ABB RobotStudio station: SD_Exe01_SWorksRStudio.rsstnx

Station SD_Exe01_SWorksRStudio (saved by RobotStudio 22.3.10190.2)
Controller CRB15000_5_95_1
  mechanical unit ROB_1: CRB15000_5_95__02, 6 joints, base frame (0, 0, 0) mm
Layout (positions relative to the parent item):
  - CRB15000_5_95__02 [mechanism, from Robots\CRB15000_5_95__02.rslib] at (0, 0, 0) mm; joint values [0.1436, 0.0868, 0.8423, 1.7766, 1.4192, 2.1968] (rad or m)
  - EF_DemoTool [mechanism] at (461.55, 153.56, 331.85) mm, rotated rx -90 ry 0 rz -6.38 deg
      TCP EF_DemoTool at (0, 0, 155) mm
      links: EF_Demo
  - part_SD_01 [part] at (485.51, 347.24, 308) mm, size 71 x 71 x 39 mm
  - table_and_fixture_140 [part, from Training Objects\propeller_table.rslib] at (292.34, 222.04, 0) mm
Attachment: EF_DemoTool is attached to CRB15000_5_95__02 / Link6
Attachment: Workobject_1 is attached to part_SD_01
Attachment: Workobject_3 is attached to table_and_fixture_140
Attachment: part_SD_01 is attached to table_and_fixture_140
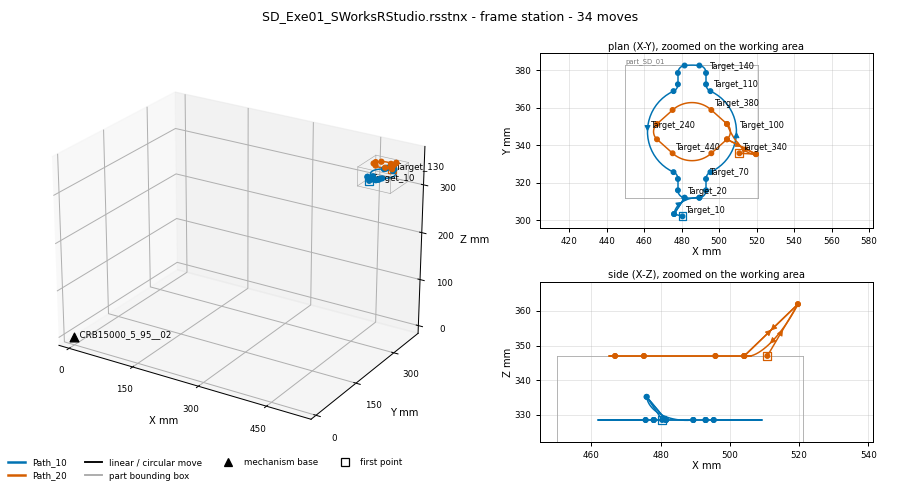
[picture p0: tool path of SD_Exe01_SWorksRStudio.rsstnx in frame station, 34 of 34 moves have a stored position in this frame; points joined in program order, loops and branches not executed]
Targets, tools, work objects and paths stored in the station, written as RAPID:
! task T_ROB1
MODULE CalibData
  PERS tooldata EF_DemoTool:=[TRUE,[[0,0,155],[1,0,0,0]],[2,[20,0,15],[1,0,0,0],0,0,0]];
  PERS wobjdata Workobject_1:=[FALSE,TRUE,"",[[485.512,347.241,308],[1,0,0,0]],[[0,0,0],[1,0,0,0]]];
  PERS wobjdata Workobject_3:=[FALSE,TRUE,"",[[485.512,347.241,308],[1,0,0,0]],[[0,0,0],[1,0,0,0]]];
ENDMODULE

! task T_ROB1
MODULE Module1
  CONST robtarget Target_10:=[[-5.055555556,-45.218263545,20.5],[0.70601133,-0.70601133,0.039344663,-0.039344663],[0,1,1,0],[9E+09,9E+09,9E+09,9E+09,9E+09,9E+09]];
  CONST robtarget Target_20:=[[-3.944444444,-35.280183645,20.5],[0.70601133,-0.70601133,0.039344663,-0.039344663],[0,1,1,0],[9E+09,9E+09,9E+09,9E+09,9E+09,9E+09]];
  CONST robtarget Target_30:=[[0,-35.5,20.5],[0.70601133,-0.70601133,0.039344663,-0.039344663],[0,1,1,0],[9E+09,9E+09,9E+09,9E+09,9E+09,9E+09]];
  CONST robtarget Target_40:=[[3.944444444,-35.280183645,20.5],[0.70601133,-0.70601133,0.039344663,-0.039344663],[0,1,1,0],[9E+09,9E+09,9E+09,9E+09,9E+09,9E+09]];
  CONST robtarget Target_50:=[[6.48142397,-33.971618352,20.5],[0.70601133,-0.70601133,0.039344663,-0.039344663],[0,1,1,0],[9E+09,9E+09,9E+09,9E+09,9E+09,9E+09]];
  CONST robtarget Target_60:=[[7.5,-31.304951685,20.5],[0.70601133,-0.70601133,0.039344663,-0.039344663],[0,1,1,0],[9E+09,9E+09,9E+09,9E+09,9E+09,9E+09]];
  CONST robtarget Target_70:=[[7.5,-25.25495001,20.5],[0.70601133,-0.70601133,0.039344663,-0.039344663],[0,1,1,0],[9E+09,9E+09,9E+09,9E+09,9E+09,9E+09]];
  CONST robtarget Target_80:=[[8.136175493,-23.090536767,20.5],[0.70601133,-0.70601133,0.039344663,-0.039344663],[0,1,1,0],[9E+09,9E+09,9E+09,9E+09,9E+09,9E+09]];
  CONST robtarget Target_90:=[[9.842342342,-21.614596855,20.5],[0.70601133,-0.70601133,0.039344663,-0.039344663],[0,1,1,0],[9E+09,9E+09,9E+09,9E+09,9E+09,9E+09]];
  CONST robtarget Target_100:=[[23.75,0,20.5],[0.70601133,-0.70601133,0.039344663,-0.039344663],[0,1,1,0],[9E+09,9E+09,9E+09,9E+09,9E+09,9E+09]];
  CONST robtarget Target_110:=[[9.842342342,21.614596855,20.5],[0.70601133,-0.70601133,0.039344663,-0.039344663],[0,1,1,0],[9E+09,9E+09,9E+09,9E+09,9E+09,9E+09]];
  CONST robtarget Target_120:=[[8.136175493,23.090536767,20.5],[0.70601133,-0.70601133,0.039344663,-0.039344663],[0,1,1,0],[9E+09,9E+09,9E+09,9E+09,9E+09,9E+09]];
  CONST robtarget Target_130:=[[7.5,25.25495001,20.5],[0.70601133,-0.70601133,0.039344663,-0.039344663],[0,1,1,0],[9E+09,9E+09,9E+09,9E+09,9E+09,9E+09]];
  CONST robtarget Target_140:=[[7.5,31.304951685,20.5],[0.70601133,-0.70601133,0.039344663,-0.039344663],[0,1,1,0],[9E+09,9E+09,9E+09,9E+09,9E+09,9E+09]];
  CONST robtarget Target_150:=[[6.48142397,33.971618352,20.5],[0.70601133,-0.70601133,0.039344663,-0.039344663],[0,1,1,0],[9E+09,9E+09,9E+09,9E+09,9E+09,9E+09]];
  CONST robtarget Target_160:=[[3.944444444,35.280183645,20.5],[0.70601133,-0.70601133,0.039344663,-0.039344663],[0,1,1,0],[9E+09,9E+09,9E+09,9E+09,9E+09,9E+09]];
  CONST robtarget Target_170:=[[0,35.5,20.5],[0.70601133,-0.70601133,0.039344663,-0.039344663],[0,1,1,0],[9E+09,9E+09,9E+09,9E+09,9E+09,9E+09]];
  CONST robtarget Target_180:=[[-3.944444444,35.280183645,20.5],[0.70601133,-0.70601133,0.039344663,-0.039344663],[0,1,1,0],[9E+09,9E+09,9E+09,9E+09,9E+09,9E+09]];
  CONST robtarget Target_190:=[[-6.48142397,33.971618352,20.5],[0.70601133,-0.70601133,0.039344663,-0.039344663],[0,1,1,0],[9E+09,9E+09,9E+09,9E+09,9E+09,9E+09]];
  CONST robtarget Target_200:=[[-7.5,31.304951685,20.5],[0.70601133,-0.70601133,0.039344663,-0.039344663],[0,1,1,0],[9E+09,9E+09,9E+09,9E+09,9E+09,9E+09]];
  CONST robtarget Target_210:=[[-7.5,25.25495001,20.5],[0.70601133,-0.70601133,0.039344663,-0.039344663],[0,1,1,0],[9E+09,9E+09,9E+09,9E+09,9E+09,9E+09]];
  CONST robtarget Target_220:=[[-8.136175493,23.090536767,20.5],[0.70601133,-0.70601133,0.039344663,-0.039344663],[0,1,1,0],[9E+09,9E+09,9E+09,9E+09,9E+09,9E+09]];
  CONST robtarget Target_230:=[[-9.842342342,21.614596855,20.5],[0.70601133,-0.70601133,0.039344663,-0.039344663],[0,1,1,0],[9E+09,9E+09,9E+09,9E+09,9E+09,9E+09]];
  CONST robtarget Target_240:=[[-23.75,0,20.5],[0.70601133,-0.70601133,0.039344663,-0.039344663],[0,1,1,0],[9E+09,9E+09,9E+09,9E+09,9E+09,9E+09]];
  CONST robtarget Target_250:=[[-9.842342342,-21.614596855,20.5],[0.70601133,-0.70601133,0.039344663,-0.039344663],[0,1,1,0],[9E+09,9E+09,9E+09,9E+09,9E+09,9E+09]];
  CONST robtarget Target_260:=[[-8.136175493,-23.090536767,20.5],[0.70601133,-0.70601133,0.039344663,-0.039344663],[0,1,1,0],[9E+09,9E+09,9E+09,9E+09,9E+09,9E+09]];
  CONST robtarget Target_270:=[[-7.5,-25.25495001,20.5],[0.70601133,-0.70601133,0.039344663,-0.039344663],[0,1,1,0],[9E+09,9E+09,9E+09,9E+09,9E+09,9E+09]];
  CONST robtarget Target_280:=[[-7.5,-31.304951685,20.5],[0.70601133,-0.70601133,0.039344663,-0.039344663],[0,1,1,0],[9E+09,9E+09,9E+09,9E+09,9E+09,9E+09]];
  CONST robtarget Target_290:=[[-6.48142397,-33.971618352,20.5],[0.70601133,-0.70601133,0.039344663,-0.039344663],[0,1,1,0],[9E+09,9E+09,9E+09,9E+09,9E+09,9E+09]];
  CONST robtarget Target_300:=[[-3.944444444,-35.280183645,20.5],[0.70601133,-0.70601133,0.039344663,-0.039344663],[0,1,1,0],[9E+09,9E+09,9E+09,9E+09,9E+09,9E+09]];
  CONST robtarget Target_310:=[[0,-35.5,20.5],[0.70601133,-0.70601133,0.039344663,-0.039344663],[0,1,1,0],[9E+09,9E+09,9E+09,9E+09,9E+09,9E+09]];
  CONST robtarget Target_320:=[[3.944444444,-35.280183645,20.5],[0.70601133,-0.70601133,0.039344663,-0.039344663],[0,1,1,0],[9E+09,9E+09,9E+09,9E+09,9E+09,9E+09]];
  CONST robtarget Target_330:=[[3.944444444,-35.280183645,30.5],[0.70601133,-0.70601133,0.039344663,-0.039344663],[0,0,0,0],[9E+09,9E+09,9E+09,9E+09,9E+09,9E+09]];
  CONST robtarget Target_20_2:=[[-9.544664008,-43.949115687,27.195284219],[0.70601133,-0.70601133,0.039344663,-0.039344663],[0,1,1,0],[9E+09,9E+09,9E+09,9E+09,9E+09,9E+09]];
  CONST robtarget Target_20_3:=[[-9.544664008,-44.003616578,27.195284219],[0.70601133,-0.70601133,0.039344663,-0.039344663],[0,1,1,0],[9E+09,9E+09,9E+09,9E+09,9E+09,9E+09]];
  CONST robtarget Target_340:=[[25.333333333,-11.553017884,39],[0.66055961,-0.66055961,-0.252311319,0.252311319],[0,0,1,0],[9E+09,9E+09,9E+09,9E+09,9E+09,9E+09]];
  CONST robtarget Target_350:=[[18.666666667,-4.099457959,39],[0.66055961,-0.66055961,-0.252311319,0.252311319],[0,0,1,0],[9E+09,9E+09,9E+09,9E+09,9E+09,9E+09]];
  CONST robtarget Target_360:=[[20.5,0,39],[0.5,-0.5,-0.5,0.5],[0,0,1,0],[9E+09,9E+09,9E+09,9E+09,9E+09,9E+09]];
  CONST robtarget Target_370:=[[18.666666667,4.099457959,39],[0.252311319,-0.252311319,-0.66055961,0.66055961],[0,-1,0,0],[9E+09,9E+09,9E+09,9E+09,9E+09,9E+09]];
  CONST robtarget Target_380:=[[10.333333333,11.553017884,39],[0.252311319,-0.252311319,-0.66055961,0.66055961],[0,-1,0,0],[9E+09,9E+09,9E+09,9E+09,9E+09,9E+09]];
  CONST robtarget Target_390:=[[0,15.5,39],[0,0,1,0],[0,-1,0,0],[9E+09,9E+09,9E+09,9E+09,9E+09,9E+09]];
  CONST robtarget Target_400:=[[-10.333333333,11.553017884,39],[0,-0.35682209,0.934172359,0],[0,0,-1,0],[9E+09,9E+09,9E+09,9E+09,9E+09,9E+09]];
  CONST robtarget Target_410:=[[-18.666666667,4.099457959,39],[0.252311319,-0.252311319,0.66055961,-0.66055961],[0,-1,0,0],[9E+09,9E+09,9E+09,9E+09,9E+09,9E+09]];
  CONST robtarget Target_420:=[[-20.5,0,39],[0,-0.707106781,0.707106781,0],[0,-1,0,0],[9E+09,9E+09,9E+09,9E+09,9E+09,9E+09]];
  CONST robtarget Target_430:=[[-18.666666667,-4.099457959,39],[0,0.934172359,-0.35682209,0],[0,0,-2,0],[9E+09,9E+09,9E+09,9E+09,9E+09,9E+09]];
  CONST robtarget Target_440:=[[-10.333333333,-11.553017884,39],[0,0.934172359,-0.35682209,0],[0,0,-2,0],[9E+09,9E+09,9E+09,9E+09,9E+09,9E+09]];
  CONST robtarget Target_450:=[[0,-15.5,39],[0,1,0,0],[0,0,-2,0],[9E+09,9E+09,9E+09,9E+09,9E+09,9E+09]];
  CONST robtarget Target_460:=[[10.333333333,-11.553017884,39],[0,0.934172359,0.35682209,0],[0,0,-3,0],[9E+09,9E+09,9E+09,9E+09,9E+09,9E+09]];
  CONST robtarget Target_470:=[[18.666666667,-4.099457959,39],[0.66055961,-0.66055961,-0.252311319,0.252311319],[0,0,-3,0],[9E+09,9E+09,9E+09,9E+09,9E+09,9E+09]];
  CONST robtarget Target_480:=[[20.5,0,39],[0,0.707106781,0.707106781,0],[0,0,-3,0],[9E+09,9E+09,9E+09,9E+09,9E+09,9E+09]];
  CONST robtarget Target_490:=[[18.666666667,4.099457959,39],[0,0.35682209,0.934172359,0],[0,0,0,0],[9E+09,9E+09,9E+09,9E+09,9E+09,9E+09]];
  CONST robtarget Target_500:=[[18.666585091,4.099494615,49.000001719],[-0.000000004,0.356822131,0.934172343,-0.000000006],[0,0,0,0],[9E+09,9E+09,9E+09,9E+09,9E+09,9E+09]];
  CONST robtarget Target_350_2:=[[34.176445897,-12.022195117,53.970253057],[0.66055961,-0.66055961,-0.252311319,0.252311319],[0,0,1,0],[9E+09,9E+09,9E+09,9E+09,9E+09,9E+09]];
  CONST robtarget Target_350_3:=[[34.176445897,-12.022195117,53.970253057],[0.66055961,-0.66055961,-0.252311319,0.252311319],[0,0,1,0],[9E+09,9E+09,9E+09,9E+09,9E+09,9E+09]];
  PROC Path_10()
    MoveJ Target_10,v1000,z100,EF_DemoTool\WObj:=Workobject_3;
    MoveL Target_20_2,v1000,z100,EF_DemoTool\WObj:=Workobject_3;
    MoveL Target_20,v1000,z100,EF_DemoTool\WObj:=Workobject_3;
    MoveC Target_30,Target_40,v1000,z100,EF_DemoTool\WObj:=Workobject_3;
    MoveC Target_50,Target_60,v1000,z100,EF_DemoTool\WObj:=Workobject_3;
    MoveL Target_70,v1000,z100,EF_DemoTool\WObj:=Workobject_3;
    MoveC Target_80,Target_90,v1000,z100,EF_DemoTool\WObj:=Workobject_3;
    MoveC Target_100,Target_110,v1000,z100,EF_DemoTool\WObj:=Workobject_3;
    MoveC Target_120,Target_130,v1000,z100,EF_DemoTool\WObj:=Workobject_3;
    MoveL Target_140,v1000,z100,EF_DemoTool\WObj:=Workobject_3;
    MoveC Target_150,Target_160,v1000,z100,EF_DemoTool\WObj:=Workobject_3;
    MoveC Target_170,Target_180,v1000,z100,EF_DemoTool\WObj:=Workobject_3;
    MoveC Target_190,Target_200,v1000,z100,EF_DemoTool\WObj:=Workobject_3;
    MoveL Target_210,v1000,z100,EF_DemoTool\WObj:=Workobject_3;
    MoveC Target_220,Target_230,v1000,z100,EF_DemoTool\WObj:=Workobject_3;
    MoveC Target_240,Target_250,v1000,z100,EF_DemoTool\WObj:=Workobject_3;
    MoveC Target_260,Target_270,v1000,z100,EF_DemoTool\WObj:=Workobject_3;
    MoveL Target_280,v1000,z100,EF_DemoTool\WObj:=Workobject_3;
    MoveC Target_290,Target_300,v1000,z100,EF_DemoTool\WObj:=Workobject_3;
    MoveL Target_20_3,v1000,z100,EF_DemoTool\WObj:=Workobject_3;
    MoveC Target_310,Target_320,v1000,z100,EF_DemoTool\WObj:=Workobject_3;
  ENDPROC
  PROC Path_20()
    MoveJ Target_340,v60,z0,EF_DemoTool\WObj:=Workobject_3;
    MoveL Target_350_2,v60,z0,EF_DemoTool\WObj:=Workobject_3;
    MoveL Target_350,v60,z0,EF_DemoTool\WObj:=Workobject_3;
    MoveC Target_360,Target_370,v60,z0,EF_DemoTool\WObj:=Workobject_3;
    MoveL Target_380,v60,z0,EF_DemoTool\WObj:=Workobject_3;
    MoveC Target_390,Target_400,v60,z0,EF_DemoTool\WObj:=Workobject_3;
    MoveL Target_410,v60,z0,EF_DemoTool\WObj:=Workobject_3;
    MoveC Target_420,Target_430,v60,z0,EF_DemoTool\WObj:=Workobject_3;
    MoveL Target_440,v60,z0,EF_DemoTool\WObj:=Workobject_3;
    MoveC Target_450,Target_460,v60,z0,EF_DemoTool\WObj:=Workobject_3;
    MoveL Target_470,v60,z0,EF_DemoTool\WObj:=Workobject_3;
    MoveL Target_350_3,v60,z0,EF_DemoTool\WObj:=Workobject_3;
    MoveC Target_480,Target_490,v60,z0,EF_DemoTool\WObj:=Workobject_3;
  ENDPROC
ENDMODULE

